DATA_BLOCK "DI_CHK_Assigned_Rout"
TITLE =%version: 0.01 % CN: 49
//History:
//This version  %created_by: nlhdl %
//              %date_created: maandag 6 juli 2015 10:44:01 %
//
//Modification History:                                   By:    Date:     Rev:
//----------------------------------------------------  -------  --------  -----
//7324: ECS-P General from the RD to RA for platform    nlHdL    06-07-15   0.01
FAMILY : General
VERSION : 0.0

"FB_CHK_Assigned_Rout"
BEGIN
END_DATA_BLOCK
